FUNCTION_BLOCK MockForwardEnumerator IMPLEMENTS I_ForwardEnumerator
VAR
	isValidState : BOOL;
	moveNextState : BOOL;
	tryGetState : BOOL;
	tryGetToState : BOOL;
END_VAR

METHOD PUBLIC Dispose
VAR_INPUT
END_VAR
END_METHOD

METHOD FB_init : BOOL
VAR_INPUT
	bInitRetains : BOOL; // if TRUE, the retain variables are initialized (warm start / cold start)
	bInCopyCode : BOOL;  // if TRUE, the instance afterwards gets moved into the copy code (online change)
	IsValidState : BOOL;
	MoveNextState : BOOL;
	TryGetState : BOOL;
	TryGetToState : BOOL;
END_VAR
THIS^.isValidState := IsValidState;
THIS^.moveNextState := MoveNextState;
THIS^.tryGetState := TryGetState;
THIS^.tryGetToState := TryGetToState;
END_METHOD

PROPERTY PUBLIC IsValid : BOOL
GET
IsValid := isValidState;
END_GET
END_PROPERTY

METHOD PUBLIC MoveNext : BOOL
MoveNext := moveNextState;
END_METHOD

METHOD PUBLIC TryGet : BOOL;
VAR_INPUT
    Destination : ANY;
END_VAR
TryGet := tryGetState;
END_METHOD

METHOD PUBLIC TryGetTo : BOOL;
VAR_INPUT
    DestinationAddress : PVOID;
    DestinationSize : UDINT;
END_VAR
TryGetTo := tryGetToState;
END_METHOD

END_FUNCTION_BLOCK

(* stored: Version 1.1.0.1, ProductVersion 3.1.4024.12
   POU MockForwardEnumerator: Id {2e6c3769-f351-4ddb-8d9d-8e5e37b6dae9}, SpecialFunc None
   Folder Constructor: Id {71773b41-cbd0-4631-9138-937346179e04}
   Method Dispose: Id {1a2fc6bc-59bb-4553-98f8-9788a903aac0}
   Method FB_init: Id {d3dc33ee-318e-4c8f-b3a3-5df67aa5fc45}
   Property IsValid: Id {9f776dc0-5e22-4124-a32e-69ffb7e8a4dd}
   Get Get: Id {d06d178d-3ea8-4500-b7e0-e1c5c8a7a326}
   Method MoveNext: Id {c2008efe-8a07-4f0a-96f0-420f056950bf}
   Method TryGet: Id {65d2b07a-f135-4612-be9e-8340f238ce6c}
   Method TryGetTo: Id {cceaf1c8-8859-4dc7-ba80-2408a6e5c28a} *)
